TEXTLIST EL2904_M_1
  1 = 'Safety output 1' | chinese: '继电器输出' | Chinese: '继电器输出'
  2 = 'Safety output 2' | chinese: '继电器输出' | Chinese: '继电器输出'
  3 = 'Safety output 3' | chinese: '继电器输出' | Chinese: '继电器输出'
  4 = 'Safety output 4' | chinese: '继电器输出' | Chinese: '继电器输出'
   = ''
END_TEXTLIST

(* stored: Version 1.1.0.1, ProductVersion 3.1.4024.11
   TextList EL2904_M_1: Id {c095b3ec-6631-40f6-89fb-185dd6ce50cf} *)
